{attribute 'linkalways'} 
{attribute 'no_explicit_call' := 'This FB is a CLASS and must be accessed using methods or properties'}
{attribute 'enable_dynamic_creation'}
FUNCTION_BLOCK _ETcVnEdgeDetectionAlgorithm EXTENDS EnumDatatypeBase
VAR
	localData : ETcVnEdgeDetectionAlgorithm;
	activeData : REFERENCE TO ETcVnEdgeDetectionAlgorithm;
	enumBaseDatatype : _DINT(localData);
END_VAR

METHOD PRIVATE AddLocalEnumeration
VAR_INPUT
	Enumeration : T_MAXSTRING;
	Value : ETcVnEdgeDetectionAlgorithm;
END_VAR
AddEnumeration(Enumeration, Value);
END_METHOD

PROPERTY PUBLIC Address : PVOID
GET
Address := ADR(activeData);
END_GET
END_PROPERTY

METHOD PUBLIC ClearReference
VAR_INPUT
END_VAR
activeData REF= localData;
SetBaseDatatypeReference();
END_METHOD

METHOD PUBLIC Clone : I_Datatype
VAR
    pClone : POINTER TO _ETcVnEdgeDetectionAlgorithm;
END_VAR
pClone := __NEW(_ETcVnEdgeDetectionAlgorithm(InitialValue := Value));
Clone := pClone^;
END_METHOD

METHOD FB_init : BOOL
VAR_INPUT
	bInitRetains : BOOL; // if TRUE, the retain variables are initialized (warm start / cold start)
	bInCopyCode : BOOL;  // if TRUE, the instance afterwards gets moved into the copy code (online change)
	InitialValue : ETcVnEdgeDetectionAlgorithm;
END_VAR
localData := InitialValue;
AddBaseDatatype(enumBaseDatatype);
ClearReference();

AddLocalEnumeration('TCVN_EDA_INTERPOLATION', ETcVnEdgeDetectionAlgorithm.TCVN_EDA_INTERPOLATION);
AddLocalEnumeration('TCVN_EDA_APPROX_ERF', ETcVnEdgeDetectionAlgorithm.TCVN_EDA_APPROX_ERF);
AddLocalEnumeration('TCVN_EDA_APPROX_GAUSSIAN', ETcVnEdgeDetectionAlgorithm.TCVN_EDA_APPROX_GAUSSIAN);
END_METHOD

PROPERTY PUBLIC Identifier : T_MAXSTRING
GET
Identifier := 'ETcVnEdgeDetectionAlgorithm';
END_GET
END_PROPERTY

METHOD IsEnumeratorValueEqual : BOOL
VAR_INPUT
	Enumerator : I_KeyValueForwardEnumerator;
END_VAR
VAR
	storedValue : ETcVnEdgeDetectionAlgorithm;
END_VAR
IF NOT Enumerator.TryGet(storedValue) THEN
	RETURN;
END_IF

IsEnumeratorValueEqual := storedValue = activeData;
END_METHOD

METHOD PUBLIC MakeReferenceTo
VAR_INPUT
	ReferenceTarget : REFERENCE TO ETcVnEdgeDetectionAlgorithm;
END_VAR
activeData REF= ReferenceTarget;
SetBaseDatatypeReference();
END_METHOD

METHOD PROTECTED SetBaseDatatypeReference
VAR_INPUT
END_VAR
enumBaseDatatype.MakeReferenceTo(activeData);
END_METHOD

PROPERTY PUBLIC Size : UDINT
GET
Size := SIZEOF(activeData);
END_GET
END_PROPERTY

METHOD TryMakeReferenceTo : BOOL
VAR_INPUT
	Target : I_Datatype;
END_VAR
VAR
	targetAsEnum : I_EnumDatatype;
	pTargetData : POINTER TO ETcVnEdgeDetectionAlgorithm;
END_VAR
IF NOT Target.TryResolveAsEnumDatatype(targetAsEnum) THEN
	RETURN;
END_IF

IF targetAsEnum.Identifier <> Identifier THEN
	RETURN;
END_IF

pTargetData := Target.Address;
activeData REF= pTargetData^;
SetBaseDatatypeReference();
TryMakeReferenceTo := TRUE;
END_METHOD

PROPERTY PUBLIC Value : ETcVnEdgeDetectionAlgorithm
GET
Value := activeData;
END_GET
SET
activeData := Value;
END_SET
END_PROPERTY

END_FUNCTION_BLOCK

(* stored: Version 1.1.0.1
   POU _ETcVnEdgeDetectionAlgorithm: Id {65301c07-07f7-450d-8627-2a58dc8b4bbb}, SpecialFunc None
   Folder Constructor: Id {ad3fcd7e-906d-4fab-a1d2-1d8ecfee0af5}
   Folder Private: Id {4195be82-8116-415d-99f1-51c98b83bda4}
   Folder Protected: Id {3af4165b-ba20-45a5-a497-59d38f6660ec}
   Method AddLocalEnumeration: Id {7c834616-99ae-49d2-ad41-478af676c002}
   Property Address: Id {46121234-43ff-4a01-9a63-bfa2b9e58786}
   Get Get: Id {27a17420-6fdd-48ca-abc1-766e5f7b80ed}
   Method ClearReference: Id {5ef7a3c8-9929-4073-882a-969eed45a33a}
   Method Clone: Id {28dff2d4-af35-4edc-accb-1bc1d45d892b}
   Method FB_init: Id {f29f6112-8b63-4c39-a665-ab6ec62c9f96}
   Property Identifier: Id {c8c38a4a-fc58-457a-abe8-29a349ccfa38}
   Get Get: Id {989285b2-27dc-4dc5-8810-192f54ad6a3c}
   Method IsEnumeratorValueEqual: Id {aea370ec-c216-422f-8dcd-37c16bd48d81}
   Method MakeReferenceTo: Id {2d1b6db8-65b2-4c01-ad89-ddf1bef47732}
   Method SetBaseDatatypeReference: Id {8fd9ab30-7d83-477e-8a5e-cd339c32bf96}
   Property Size: Id {61a1d39c-27c8-4051-8da8-313141372e37}
   Get Get: Id {154bfc2a-7fc2-4fd0-87ab-b61117824e4f}
   Method TryMakeReferenceTo: Id {c01cc88a-898b-421a-80e2-efb8597e0981}
   Property Value: Id {2d1fd32d-da42-4d82-9952-ac1f6c0195f5}
   Get Get: Id {0009866a-152f-4f5d-bcfa-5925239deb1f}
   Set Set: Id {b3edd817-5cad-4dee-9836-08fe0708a513} *)
